// TIA Portal V20 export
DATA_BLOCK "HandyReader_UnUsed"   // DB348
// stored: MemoryReserve 100, Namespace Unit1
   VAR
      ClientPara : Struct
         REQ : Bool;
         DISCONNECT : Bool;
         MB_MODE : USInt := 103;
         MB_DATA_ADDR : UDInt := 7000;
         MB_DATA_LEN : UInt := 25;
         MB_DATA_PTR : Array[0..50] of Char;
         connectParaClient : TCON_IP_v4;
         DONE { S7_SetPoint := 'True'} : Bool;
         BUSY : Bool;
         ERROR { S7_SetPoint := 'True'} : Bool;
         STATUS { S7_SetPoint := 'True'} : Word;
      END_STRUCT;
      BCR_Read : String;
      BCR_Read_Convert : Array[0..30] of Char;
   END_VAR
BEGIN
   ClientPara.connectParaClient.InterfaceId := 120;
   ClientPara.connectParaClient.ID := 16#1;
   ClientPara.connectParaClient.ConnectionType := 11;
   ClientPara.connectParaClient.ActiveEstablished := true;
   ClientPara.connectParaClient.RemoteAddress.ADDR[1] := 120;
   ClientPara.connectParaClient.RemoteAddress.ADDR[2] := 43;
   ClientPara.connectParaClient.RemoteAddress.ADDR[3] := 138;
   ClientPara.connectParaClient.RemoteAddress.ADDR[4] := 105;
   ClientPara.connectParaClient.RemotePort := 502;
   ClientPara.connectParaClient.LocalPort := 0;
END_DATA_BLOCK
